// TIA Portal project "AMATROL_STATION_2" (V16)

(* hardware
DEVICE "S7300/ET200M station_1"  S7-300 station
   slot 0: "Rail_0"  Rail  6ES7 390-1***0-0AA0
   slot 2: "PLC_1"  CPU 314C-2 DP  6ES7 314-6CH04-0AB0  V3.3
      slot 0: "MPI interface_1"  MPI
      slot 1: "DP interface_1"  DP
      slot 2: "DI 24/DO 16_1"  DI24/DO16
      slot 3: "AI 5/AO 2_1"  AI5/AO2
      slot 4: "Count_1"  Counter
      slot 5: "Positioning_1"  Positioning
*)

// ===== PLC "PLC_1"  CPU 314C-2 DP =====

VAR_GLOBAL   // PLC tag table "INPUTS AND OUTPUTS"
   "S3_START" AT %I0.0 : Bool;
   "S4_STOP" AT %I0.1 : Bool;
   "S5_EMERGENCY STOP" AT %I0.2 : Bool;
   "S2_OUTPUT_POWER" AT %I0.3 : Bool;
   "3B1_REJECT_CYLINDER_RETRACTED" AT %I1.2 : Bool;
   "3B2_REJECT_CYLINDER_EXTENDED" AT %I1.3 : Bool;
   "1B1_TRANSFER_CYLINDER_RETRACTED" AT %I1.4 : Bool;
   "1B2_TRANSFER_CYLINDER_EXTENDED" AT %I1.5 : Bool;
   "4S2_TRAVERSE_END" AT %I1.6 : Bool;
   "4S1_TRAVERSE_START" AT %I1.7 : Bool;
   "B2" AT %I2.2 : Bool;   // PART IN HEIGHT MEASURING POSITION(INDUCTIVE SENSOR)
   "B3" AT %I2.3 : Bool;   // PART HEIGHT READING(ULTRASONIC SENSOR)
   "B1" AT %I2.4 : Bool;   // PART NOT DETECTED (LIGHT SENSOR )
   "H3_GREEN" AT %Q4.0 : Bool;
   "3M1_EXTEND_REJECT_CYLINDER" AT %Q4.5 : Bool;
   "1M1_EXTEND_TRANSFER_CYLINDER" AT %Q4.6 : Bool;
   "1M2_RETRACT_TRANSFER_CYLINDER" AT %Q4.7 : Bool;
   "K4_MOTOR_FORWARD" AT %Q5.0 : Bool;
   "K5_MOTOR_REVERSE" AT %Q5.1 : Bool;
   "2M1_EXTEND_LIFT_CYLINDER" AT %Q5.6 : Bool;
   "S6_RESET" AT %I1.0 : Bool;
   "S6_AUTO" AT %I1.1 : Bool;
END_VAR

DATA_BLOCK "STEPS"   // DB1
{ S7_Optimized_Access := 'FALSE' }
VERSION : 0.1
   VAR
      Current_step : Int;
   END_VAR
BEGIN
END_DATA_BLOCK

ORGANIZATION_BLOCK "Main"   // OB1, LAD
TITLE = "Main Program Sweep (Cycle)"
{ S7_Optimized_Access := 'FALSE' }
VERSION : 0.1
   VAR_TEMP
      OB1_EV_CLASS : Byte;   // Bits 0-3 = 1 (Coming event), Bits 4-7 = 1 (Event class 1)
      OB1_SCAN_1 : Byte;   // 1 (Cold restart scan 1 of OB 1), 3 (Scan 2-n of OB 1)
      OB1_PRIORITY : Byte;   // Priority of OB Execution
      OB1_OB_NUMBR : Byte;   // 1 (Organization block 1, OB1)
      OB1_RESERVED_1 : Byte;   // Reserved for system
      OB1_RESERVED_2 : Byte;   // Reserved for system
      OB1_PREV_CYCLE : Int;   // Cycle time of previous OB1 scan (milliseconds)
      OB1_MIN_CYCLE : Int;   // Minimum cycle time of OB1 (milliseconds)
      OB1_MAX_CYCLE : Int;   // Maximum cycle time of OB1 (milliseconds)
      OB1_DATE_TIME : Date_And_Time;   // Date and time OB1 started
   END_VAR
   VAR_TEMP   // added for the SCL form of the ladder/FBD networks
      _w1 : Bool;
   END_VAR
BEGIN

REGION Network 1
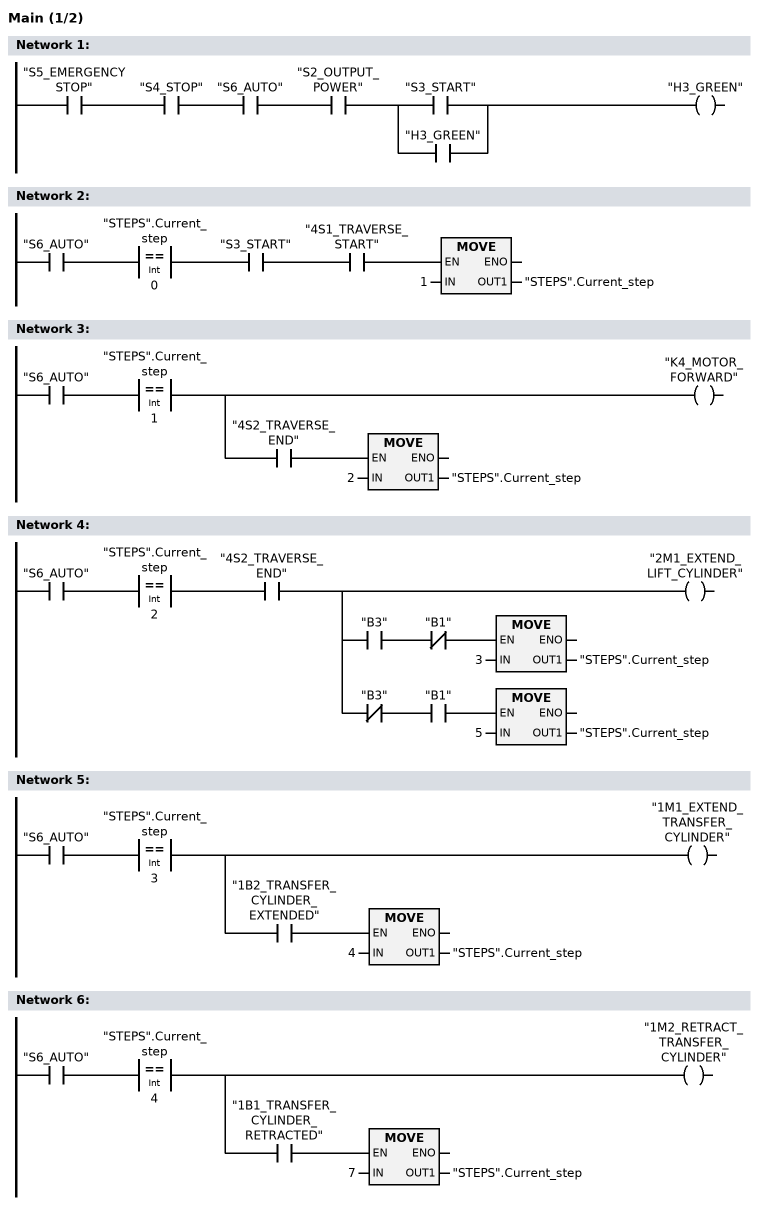
   RUNG wire#powerrail
      Contact( "S5_EMERGENCY STOP" )
      Contact( "S4_STOP" )
      Contact( "S6_AUTO" )
      Contact( "S2_OUTPUT_POWER" )
      wire#w1
      Contact( "S3_START" )
      wire#w2
      Coil( "H3_GREEN" )
   END_RUNG
   RUNG wire#w1
      Contact( "H3_GREEN" )
   END_RUNG wire#w2
   // the same network as SCL:
   "H3_GREEN" := "S5_EMERGENCY STOP" AND "S4_STOP" AND "S6_AUTO" AND "S2_OUTPUT_POWER" AND ("S3_START" OR "H3_GREEN");
END_REGION

REGION Network 2
   RUNG wire#powerrail
      Contact( "S6_AUTO" )
      { S7_Templates := "SrcType := Int" } EQ_Contact(in1 := "STEPS".Current_step, in2 := 0)
      Contact( "S3_START" )
      Contact( "4S1_TRAVERSE_START" )
      { S7_GenerateENO := "TRUE" } Move(in := 1, out1 => "STEPS".Current_step)
   END_RUNG
   // the same network as SCL:
   IF "S6_AUTO" AND ("STEPS".Current_step = 0) AND "S3_START" AND "4S1_TRAVERSE_START" THEN
       "STEPS".Current_step := 1;
   END_IF;
END_REGION

REGION Network 3
   RUNG wire#powerrail
      Contact( "S6_AUTO" )
      { S7_Templates := "SrcType := Int" } EQ_Contact(in1 := "STEPS".Current_step, in2 := 1)
      wire#w1
      Coil( "K4_MOTOR_FORWARD" )
   END_RUNG
   RUNG wire#w1
      Contact( "4S2_TRAVERSE_END" )
      { S7_GenerateENO := "TRUE" } Move(in := 2, out1 => "STEPS".Current_step)
   END_RUNG
   // the same network as SCL:
   "K4_MOTOR_FORWARD" := "S6_AUTO" AND ("STEPS".Current_step = 1);
   IF "K4_MOTOR_FORWARD" AND "4S2_TRAVERSE_END" THEN "STEPS".Current_step := 2; END_IF;
END_REGION

REGION Network 4
   RUNG wire#powerrail
      Contact( "S6_AUTO" )
      { S7_Templates := "SrcType := Int" } EQ_Contact(in1 := "STEPS".Current_step, in2 := 2)
      Contact( "4S2_TRAVERSE_END" )
      wire#w1
      Coil( "2M1_EXTEND_LIFT_CYLINDER" )
   END_RUNG
   RUNG wire#w1
      Contact( "B3" )
      I_Contact( "B1" )
      { S7_GenerateENO := "TRUE" } Move(in := 3, out1 => "STEPS".Current_step)
   END_RUNG
   RUNG wire#w1
      I_Contact( "B3" )
      Contact( "B1" )
      { S7_GenerateENO := "TRUE" } Move(in := 5, out1 => "STEPS".Current_step)
   END_RUNG
   // the same network as SCL:
   "2M1_EXTEND_LIFT_CYLINDER" := "S6_AUTO" AND ("STEPS".Current_step = 2) AND "4S2_TRAVERSE_END";
   IF "2M1_EXTEND_LIFT_CYLINDER" AND "B3" AND NOT "B1" THEN "STEPS".Current_step := 3; END_IF;
   IF "2M1_EXTEND_LIFT_CYLINDER" AND NOT "B3" AND "B1" THEN "STEPS".Current_step := 5; END_IF;
END_REGION

REGION Network 5
   RUNG wire#powerrail
      Contact( "S6_AUTO" )
      { S7_Templates := "SrcType := Int" } EQ_Contact(in1 := "STEPS".Current_step, in2 := 3)
      wire#w1
      Coil( "1M1_EXTEND_TRANSFER_CYLINDER" )
   END_RUNG
   RUNG wire#w1
      Contact( "1B2_TRANSFER_CYLINDER_EXTENDED" )
      { S7_GenerateENO := "TRUE" } Move(in := 4, out1 => "STEPS".Current_step)
   END_RUNG
   // the same network as SCL:
   "1M1_EXTEND_TRANSFER_CYLINDER" := "S6_AUTO" AND ("STEPS".Current_step = 3);
   IF "1M1_EXTEND_TRANSFER_CYLINDER" AND "1B2_TRANSFER_CYLINDER_EXTENDED" THEN
       "STEPS".Current_step := 4;
   END_IF;
END_REGION

REGION Network 6
   RUNG wire#powerrail
      Contact( "S6_AUTO" )
      { S7_Templates := "SrcType := Int" } EQ_Contact(in1 := "STEPS".Current_step, in2 := 4)
      wire#w1
      Coil( "1M2_RETRACT_TRANSFER_CYLINDER" )
   END_RUNG
   RUNG wire#w1
      Contact( "1B1_TRANSFER_CYLINDER_RETRACTED" )
      { S7_GenerateENO := "TRUE" } Move(in := 7, out1 => "STEPS".Current_step)
   END_RUNG
   // the same network as SCL:
   "1M2_RETRACT_TRANSFER_CYLINDER" := "S6_AUTO" AND ("STEPS".Current_step = 4);
   IF "1M2_RETRACT_TRANSFER_CYLINDER" AND "1B1_TRANSFER_CYLINDER_RETRACTED" THEN
       "STEPS".Current_step := 7;
   END_IF;
END_REGION

REGION Network 7
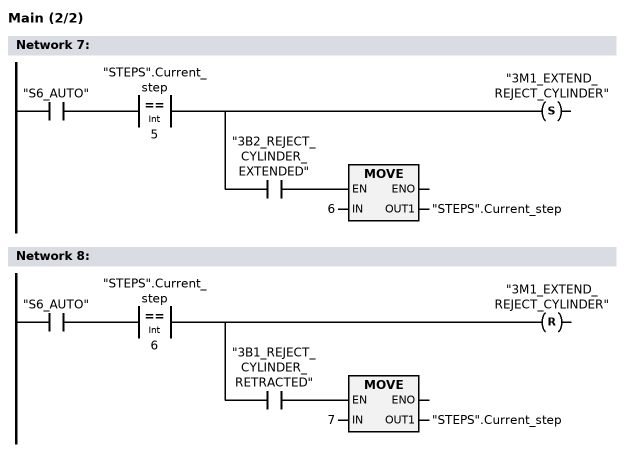
   RUNG wire#powerrail
      Contact( "S6_AUTO" )
      { S7_Templates := "SrcType := Int" } EQ_Contact(in1 := "STEPS".Current_step, in2 := 5)
      wire#w1
      S_Coil( "3M1_EXTEND_REJECT_CYLINDER" )
   END_RUNG
   RUNG wire#w1
      Contact( "3B2_REJECT_CYLINDER_EXTENDED" )
      { S7_GenerateENO := "TRUE" } Move(in := 6, out1 => "STEPS".Current_step)
   END_RUNG
   // the same network as SCL:
   #_w1 := "S6_AUTO" AND ("STEPS".Current_step = 5);
   IF #_w1 THEN "3M1_EXTEND_REJECT_CYLINDER" := TRUE; END_IF;
   IF #_w1 AND "3B2_REJECT_CYLINDER_EXTENDED" THEN "STEPS".Current_step := 6; END_IF;
END_REGION

REGION Network 8
   RUNG wire#powerrail
      Contact( "S6_AUTO" )
      { S7_Templates := "SrcType := Int" } EQ_Contact(in1 := "STEPS".Current_step, in2 := 6)
      wire#w1
      R_Coil( "3M1_EXTEND_REJECT_CYLINDER" )
   END_RUNG
   RUNG wire#w1
      Contact( "3B1_REJECT_CYLINDER_RETRACTED" )
      { S7_GenerateENO := "TRUE" } Move(in := 7, out1 => "STEPS".Current_step)
   END_RUNG
   // the same network as SCL:
   #_w1 := "S6_AUTO" AND ("STEPS".Current_step = 6);
   IF #_w1 THEN "3M1_EXTEND_REJECT_CYLINDER" := FALSE; END_IF;
   IF #_w1 AND "3B1_REJECT_CYLINDER_RETRACTED" THEN "STEPS".Current_step := 7; END_IF;
END_REGION
END_ORGANIZATION_BLOCK